FUNCTION_BLOCK FB_TempSensor_Test EXTENDS FB_TestSuite
VAR
END_VAR

Initialization();
ValidTemperatureReading();
UpdateRefreshesTemparature();
DetectOutOfRange();
InvalidReadingDoesNotUpdateGoodValue();
SensorRecoversFromFault();

METHOD DetectOutOfRange : REFERENCE TO FB_Test
VAR_INPUT
END_VAR
END_METHOD

METHOD Initialization : REFERENCE TO FB_Test
VAR_INPUT
END_VAR
END_METHOD

METHOD InvalidReadingDoesNotUpdateGoodValue : REFERENCE TO FB_Test
VAR_INPUT
END_VAR
END_METHOD

METHOD SensorRecoversFromFault : REFERENCE TO FB_Test
VAR_INPUT
END_VAR
END_METHOD

METHOD UpdateRefreshesTemparature : REFERENCE TO FB_Test
VAR_INPUT
END_VAR
END_METHOD

METHOD ValidTemperatureReading : REFERENCE TO FB_Test
VAR_INPUT
END_VAR
END_METHOD

END_FUNCTION_BLOCK

(* stored: Version 1.1.0.1
   POU FB_TempSensor_Test: Id {e8bb7e7a-3fea-489c-a564-220668290bd2}, SpecialFunc None
   Method DetectOutOfRange: Id {6d97aa0d-1b5a-4f8c-a699-883387b60166}
   Method Initialization: Id {38bb8039-0a63-42ae-9c6d-64297e97eb52}
   Method InvalidReadingDoesNotUpdateGoodValue: Id {48ef7f18-f1a5-45d4-b62b-3b54d2e7d744}
   Method SensorRecoversFromFault: Id {705e107a-dc2a-47a4-b4a3-4b7e56a3c614}
   Method UpdateRefreshesTemparature: Id {5220d095-55f8-42b1-b8ad-86a159e77a26}
   Method ValidTemperatureReading: Id {9c051db7-d449-4d7b-a34c-49c1aa8c48de} *)
